// TIA Portal project "On_Dinh_Ap_Suat" (V16)

(* hardware
DEVICE "S71500/ET200MP station_1"  S7-1500 station
   slot 0: "Rail_0"  Rack  6ES7 590-1***0-0AA0
   slot 1: "PLC_1"  CPU 1511-1 PN  6ES7 511-1AK02-0AB0  V2.8
      slot 3: "CPU display_1"  6ES7591-1AA00-0AA0
      slot 32768: "PROFINET interface_1"  X1
         slot 32769: "Port_1"  X1 P1
         slot 32770: "Port_2"  X1 P2
      slot 34817: "Virtual CP interface port_1"  Virtual CP interface port  Virtual CP interface port
   slot 2: "DI 32x24VDC HF_1"  DI 32x24VDC HF  6ES7 521-1BL00-0AB0  V2.2
   slot 3: "DQ 32x24VDC/0.5A HF_1"  DQ 32x24VDC/0.5A HF  6ES7 522-1BL01-0AB0  V1.1
   slot 4: "AQ 4xU/I ST_1"  AQ 4xU/I ST  6ES7 532-5HD00-0AB0  V2.2
DEVICE "HMI_1"  KTP700 Basic PN
   slot 0: "HMI_1"  KTP700 Basic PN  6AV2 123-2GB03-0AX0  16.0.0.0
   slot 1: "HMI_RT_1"  KTP700 Basic PN  6AV2 123-2GB03-0AX0  16.0.0.0
   slot 5: "HMI_1.IE_CP_1"  PROFINET Interface  16.0.0.0
      slot 1: "PROFINET Interface_1"  PROFINET Interface
         slot 1: "Port_1"  Port
*)

// ===== PLC "PLC_1"  CPU 1511-1 PN =====

VAR_GLOBAL   // PLC tag table "Default tag table"
   "start" AT %I0.5 : Bool;
   "stop" AT %I1.6 : Bool;
   "Tag_1" AT %M0.2 : Bool;
END_VAR

VAR_GLOBAL   // PLC tag table "I_input"
   "S_Pressure" AT %IW82 : Word;
END_VAR

VAR_GLOBAL   // PLC tag table "M_TG"
   "Temp_1" AT %MD20 : Real;
   "PV_Pressure" AT %MD24 : Real;
   "Temp_2" AT %MD28 : Real;
   "Temp_3" AT %MD32 : Real;
   "Run/Stop_Invt" AT %M0.0 : Bool;
   "On/Off" AT %M0.1 : Bool;
   "GAIN" AT %MD36 : Real;
   "TI" AT %MD40 : Real;
   "TD" AT %MD44 : Real;
END_VAR

VAR_GLOBAL   // PLC tag table "Q_Output"
   "PID_To_INVT" AT %QW50 : Int;
   "START_INVT" AT %Q1.1 : Bool;
END_VAR

DATA_BLOCK "PID"   // DB2
{ S7_Optimized_Access := 'FALSE' }
VERSION : 0.1
   VAR
      Setpoint : Real;
      PID_Output : Word;
      PID_Freq_Hz : Real;
   END_VAR
BEGIN
END_DATA_BLOCK

DATA_BLOCK "DB_WebSever"   // DB3
{ S7_Optimized_Access := 'FALSE' }
VERSION : 0.1
   VAR
      WebSite_Setpoint : Real;
      WebSite_PID_Output : Real;
      WebSite_PID_Freq_Hz : Int;
      WebSite_PV_Pressure : Real;
      WebSite_PID_Gain : Real;
      WebSite_PID_Ti : Real;
      WebSite_PID_Td : Real;
      WebSite_On_Off : Bool;
      sql_insert_Trigger : Bool;
      WebSite_Setting_Setpoint : Real;
      WebSite_Setting_Gain : Real;
      WebSite_Setting_Ti : Real;
      WebSite_Setting_Td : Real;
   END_VAR
BEGIN
END_DATA_BLOCK

FUNCTION "FTinhASThucTe" : Void   // FC1, LAD
{ S7_Optimized_Access := 'TRUE' }
VERSION : 0.1
BEGIN

REGION Network 1
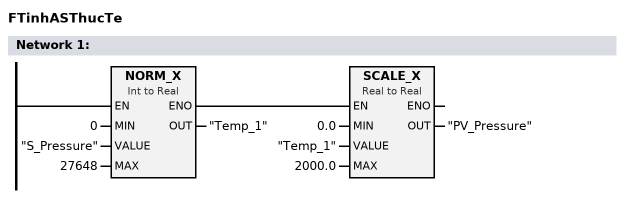
   RUNG wire#powerrail
      { S7_Templates := "[SrcType := Int, DestType := Real]" } Normalize(min := 0, value := "S_Pressure", max := 27648, out => "Temp_1")
      { S7_Templates := "[SrcType := Real, DestType := Real]" } Scale(min := 0.0, value := "Temp_1", max := 2000.0, out => "PV_Pressure")
   END_RUNG
   // the same network as SCL:
   "Temp_1" := NORM_X(MIN := 0, VALUE := "S_Pressure", MAX := 27648);
   "PV_Pressure" := SCALE_X(MIN := 0.0, VALUE := "Temp_1", MAX := 2000.0);
END_REGION
END_FUNCTION

FUNCTION "PID_To_Freq" : Void   // FC2, LAD
{ S7_Optimized_Access := 'TRUE' }
VERSION : 0.1
BEGIN

REGION Network 1
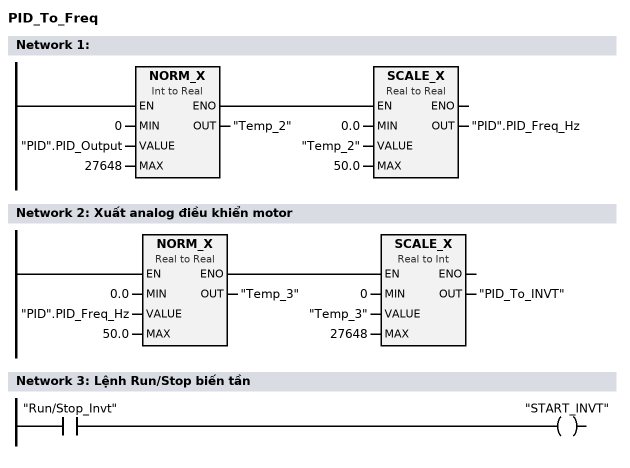
   RUNG wire#powerrail
      { S7_Templates := "[SrcType := Int, DestType := Real]" } Normalize(min := 0, value := "PID".PID_Output, max := 27648, out => "Temp_2")
      { S7_Templates := "[SrcType := Real, DestType := Real]" } Scale(min := 0.0, value := "Temp_2", max := 50.0, out => "PID".PID_Freq_Hz)
   END_RUNG
   // the same network as SCL:
   "Temp_2" := NORM_X(MIN := 0, VALUE := "PID".PID_Output, MAX := 27648);
   "PID".PID_Freq_Hz := SCALE_X(MIN := 0.0, VALUE := "Temp_2", MAX := 50.0);
END_REGION

REGION Network 2: Xuất analog điều khiển motor
   RUNG wire#powerrail
      { S7_Templates := "[SrcType := Real, DestType := Real]" } Normalize(min := 0.0, value := "PID".PID_Freq_Hz, max := 50.0, out => "Temp_3")
      { S7_Templates := "[SrcType := Real, DestType := Int]" } Scale(min := 0, value := "Temp_3", max := 27648, out => "PID_To_INVT")
   END_RUNG
   // the same network as SCL:
   "Temp_3" := NORM_X(MIN := 0.0, VALUE := "PID".PID_Freq_Hz, MAX := 50.0);
   "PID_To_INVT" := SCALE_X(MIN := 0, VALUE := "Temp_3", MAX := 27648);
END_REGION

REGION Network 3: Lệnh Run/Stop biến tần
   RUNG wire#powerrail
      Contact( "Run/Stop_Invt" )
      Coil( "START_INVT" )
   END_RUNG
   // the same network as SCL:
   "START_INVT" := "Run/Stop_Invt";
END_REGION
END_FUNCTION

FUNCTION "FC_TranformData" : Void   // FC3, LAD
{ S7_Optimized_Access := 'TRUE' }
VERSION : 0.1
BEGIN

REGION Network 1
   // PID
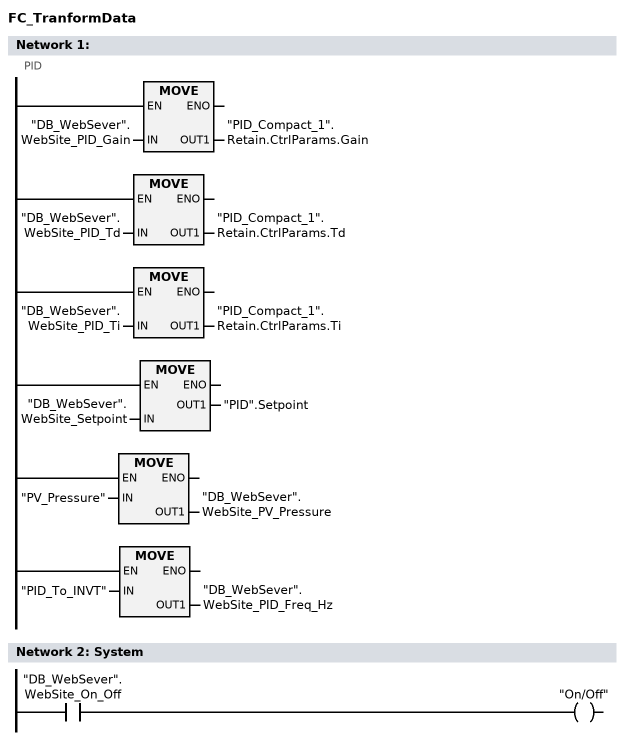
   RUNG wire#powerrail
      Move(in := "DB_WebSever".WebSite_PID_Gain, out1 => "PID_Compact_1".Retain.CtrlParams.Gain)
   END_RUNG
   RUNG wire#powerrail
      Move(in := "DB_WebSever".WebSite_PID_Td, out1 => "PID_Compact_1".Retain.CtrlParams.Td)
   END_RUNG
   RUNG wire#powerrail
      Move(in := "DB_WebSever".WebSite_PID_Ti, out1 => "PID_Compact_1".Retain.CtrlParams.Ti)
   END_RUNG
   RUNG wire#powerrail
      Move(in := "DB_WebSever".WebSite_Setpoint, out1 => "PID".Setpoint)
   END_RUNG
   RUNG wire#powerrail
      Move(in := "PV_Pressure", out1 => "DB_WebSever".WebSite_PV_Pressure)
   END_RUNG
   RUNG wire#powerrail
      Move(in := "PID_To_INVT", out1 => "DB_WebSever".WebSite_PID_Freq_Hz)
   END_RUNG
   // the same network as SCL:
   "PID_Compact_1".Retain.CtrlParams.Gain := "DB_WebSever".WebSite_PID_Gain;
   "PID_Compact_1".Retain.CtrlParams.Td := "DB_WebSever".WebSite_PID_Td;
   "PID_Compact_1".Retain.CtrlParams.Ti := "DB_WebSever".WebSite_PID_Ti;
   "PID".Setpoint := "DB_WebSever".WebSite_Setpoint;
   "DB_WebSever".WebSite_PV_Pressure := "PV_Pressure";
   "DB_WebSever".WebSite_PID_Freq_Hz := "PID_To_INVT";
END_REGION

REGION Network 2: System
   RUNG wire#powerrail
      Contact( "DB_WebSever".WebSite_On_Off )
      Coil( "On/Off" )
   END_RUNG
   // the same network as SCL:
   "On/Off" := "DB_WebSever".WebSite_On_Off;
END_REGION
END_FUNCTION

ORGANIZATION_BLOCK "Main"   // OB1, LAD, ProgramCycle
TITLE = "Main Program Sweep (Cycle)"
{ S7_Optimized_Access := 'TRUE' }
VERSION : 0.1
   VAR_INPUT
      Initial_Call : Bool;   // Initial call of this OB
      Remanence : Bool;   // =True, if remanent data are available
   END_VAR
   VAR_TEMP   // added for the SCL form of the ladder/FBD networks
      _w1 : Bool;
   END_VAR
BEGIN

REGION Network 1
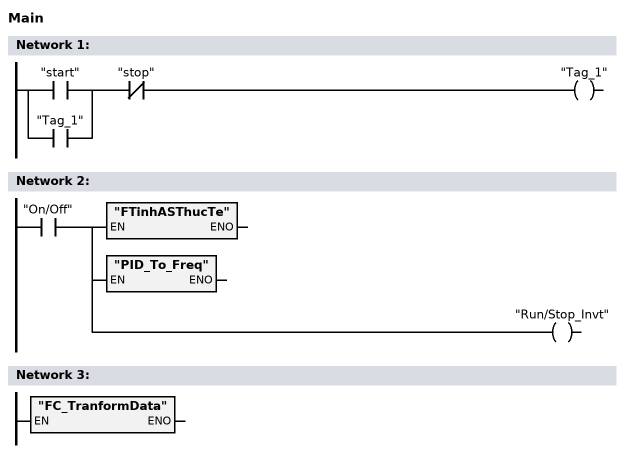
   RUNG wire#powerrail
      Contact( "start" )
      wire#w1
      I_Contact( "stop" )
      Coil( "Tag_1" )
   END_RUNG
   RUNG wire#powerrail
      Contact( "Tag_1" )
   END_RUNG wire#w1
   // the same network as SCL:
   "Tag_1" := ("start" OR "Tag_1") AND NOT "stop";
END_REGION

REGION Network 2
   RUNG wire#powerrail
      Contact( "On/Off" )
      wire#w1
      "FTinhASThucTe"()
   END_RUNG
   RUNG wire#w1
      "PID_To_Freq"()
   END_RUNG
   RUNG wire#w1
      Coil( "Run/Stop_Invt" )
   END_RUNG
   // the same network as SCL:
   #_w1 := "On/Off";
   IF #_w1 THEN
       "FTinhASThucTe"();
       "PID_To_Freq"();
   END_IF;
   "Run/Stop_Invt" := #_w1;
END_REGION

REGION Network 3
   RUNG wire#powerrail
      "FC_TranformData"()
   END_RUNG
   // the same network as SCL:
   "FC_TranformData"();
END_REGION
END_ORGANIZATION_BLOCK

ORGANIZATION_BLOCK "Cyclic interrupt"   // OB30, LAD, CyclicInterrupt
{ S7_Optimized_Access := 'TRUE' }
VERSION : 0.1
   VAR_INPUT
      Initial_Call : Bool;   // Initial call of this OB
      Event_Count : Int;   // Events discarded
   END_VAR
BEGIN

REGION Network 1
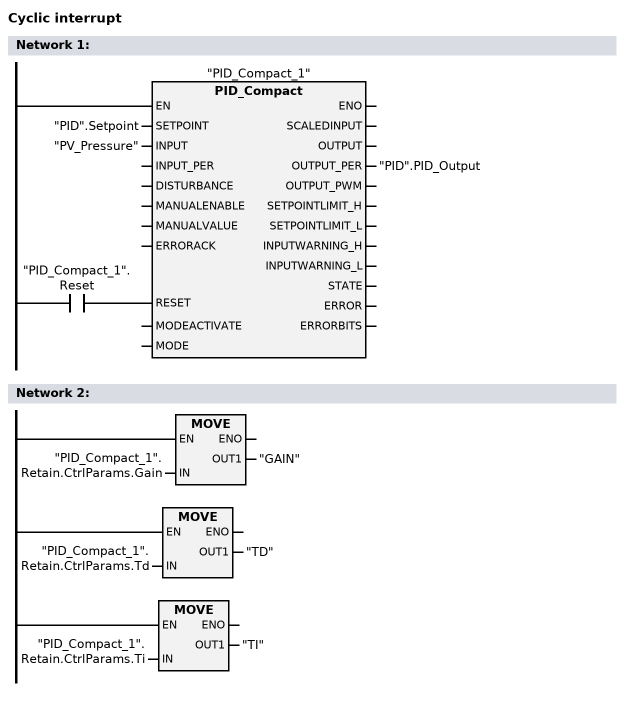
   "PID_Compact_1"(Setpoint := "PID".Setpoint,   // PID_Compact
                   Input := "PV_Pressure",
                   Reset := "PID_Compact_1".Reset,
                   Output_PER => "PID".PID_Output);
END_REGION

REGION Network 2
   RUNG wire#powerrail
      Move(in := "PID_Compact_1".Retain.CtrlParams.Gain, out1 => "GAIN")
   END_RUNG
   RUNG wire#powerrail
      Move(in := "PID_Compact_1".Retain.CtrlParams.Td, out1 => "TD")
   END_RUNG
   RUNG wire#powerrail
      Move(in := "PID_Compact_1".Retain.CtrlParams.Ti, out1 => "TI")
   END_RUNG
   // the same network as SCL:
   "GAIN" := "PID_Compact_1".Retain.CtrlParams.Gain;
   "TD" := "PID_Compact_1".Retain.CtrlParams.Td;
   "TI" := "PID_Compact_1".Retain.CtrlParams.Ti;
END_REGION
END_ORGANIZATION_BLOCK

(* ===== HMI "HMI_RT_1" =====
system functions are stored by id; their names below are inferred from use
connection "HMI_Connection_1": ETHERNET, SMART_S7_1500_OMS

HMI tags "Default tag table"
   "On/Off" : Bool = PLC "On/Off" AT %M0.1, 1 s
   "SetPoint" : Real = PLC PID.Setpoint AT %DB2.DBD0, 1 s
   "PV_Pressure" : Real = PLC PV_Pressure AT %MD24, 1 s
   "PID_output" : Real = PLC PID.PID_Freq_Hz AT %DB2.DBD6, 1 s
   "GAIN" : Real = PLC GAIN AT %MD36, 1 s
   "TI" : Real = PLC TI AT %MD40, 1 s
   "TD" : Real = PLC TD AT %MD44, 1 s

screen "Root screen" 800x480, template "Template_1"
   TrendView "Trend view_1" at 161,5 size 635x415
   Switch "Switch_1" at 15,40 size 96x32; CaptionText 'Switch'; TextOff 'OFF'; TextOn 'ON'
      ProcessValue <- "On/Off"
      on SwitchOn: SetBit("On/Off")
      on SwitchOff: ResetBit("On/Off")
   Rectangle "Rectangle_1" at 15,22 size 96x12
      Appearance <- "On/Off"
   TextField "Text field_7" at 110,354 size 43x23; Text 'SP'
   TextField "Text field_8" at 110,386 size 74x23; Text 'PRES'
   IOField "I/O field_4" at 259,429 size 96x39; FormatPattern s999.999
      ProcessValue <- "GAIN"
   TextField "Text field_9" at 202,440 size 49x23; Text 'GAIN'
   IOField "I/O field_5" at 432,429 size 96x39; FormatPattern s999.999
      ProcessValue <- "TI"
   TextField "Text field_10" at 387,440 size 49x23; Text 'TI'
   IOField "I/O field_6" at 605,429 size 96x39; FormatPattern s999.999
      ProcessValue <- "TD"
   TextField "Text field_11" at 560,440 size 49x23; Text 'TD'
   IOField "I/O field_1" at 15,120 size 96x32
      ProcessValue <- "SetPoint"
   TextField "Text field_1" at 111,125 size 47x23; Text '(kPA)'
   TextField "Text field_4" at 15,92 size 102x23; Text 'SETPOINT'
   IOField "I/O field_2" at 15,202 size 96x32
      ProcessValue <- "PV_Pressure"
   TextField "Text field_2" at 111,207 size 49x23; Text '(kPA)'
   TextField "Text field_5" at 15,173 size 112x23; Text 'PRESSERET'
   IOField "I/O field_3" at 15,286 size 96x32
      ProcessValue <- "PID_output"
   TextField "Text field_3" at 111,291 size 43x23; Text '(Hz)'
   TextField "Text field_6" at 15,256 size 102x23; Text 'OUTPUT'

screen "Root screen_1" 800x480, template "Template_1"
   TextField "Text field_7" at 110,354 size 43x23; Text 'SP'
   TextField "Text field_8" at 110,386 size 74x23; Text 'PRES'
   TextField "Text field_9" at 202,440 size 49x23; Text 'GAIN'
   TextField "Text field_10" at 387,440 size 49x23; Text 'TI'
   TextField "Text field_11" at 560,440 size 49x23; Text 'TD'
   TextField "Text field_1" at 111,125 size 47x23; Text '(kPA)'
   TextField "Text field_4" at 15,92 size 107x24; Text 'SETPOINT'
   TextField "Text field_2" at 111,207 size 49x23; Text '(kPA)'
   TextField "Text field_5" at 15,173 size 112x23; Text 'PRESSERET'
   TextField "Text field_3" at 111,291 size 43x23; Text '(Hz)'
   TextField "Text field_6" at 15,256 size 102x23; Text 'OUTPUT'
*)